// TIA Portal V20 export
TYPE "UDT_VALVE"
TITLE = DEMO
// Autor: SICAR / Autor: Tesla
   STRUCT
      Auto_Work : Bool;   // Cmd To Move Valve To Work / Cmd 到 移动 汽阀 到 工作位
      Auto_Home : Bool;   // Cmd To Move Valve To Home / Cmd 到 移动 汽阀 到 原位
      At_Work : Bool;   // Status At Work / 状态 在 工作位
      At_Home : Bool;   // Status At Home / 状态 在 原位
      Enable_Work : Bool;   // interlock to move valve to Work / 互锁 到 移动 汽阀 到 工作位
      Enable_Home : Bool;   // interlock to move valve to Home / 互锁 到 移动 汽阀 到 原位
      General_Alarm : Bool;
      Known_Position : Bool;
      Position : "VALVE_POSITION_UDT";   // Feedback from Sensors / 反馈 从 Sensors
   END_STRUCT;
END_TYPE
